// TIA Portal V19 export
FUNCTION "M_CmpGTE" : Bool   // FC43, LAD
TITLE = Module compare GREATHER THAN EQUAL / Module compare Greater than equal
// stored: Access Published, SetENOAutomatically false
   VAR_INPUT
      Xa : LReal;
      Xb : LReal;
      MODULE : LReal;
   END_VAR
BEGIN

REGION Network 1 (SCL): Xa >= Xb return TRUE / Main
   #M_CmpGTE := "M_PosAMinusPosB"(PosA := #Xa, PosB := #Xb, MODULE := #MODULE) >= 0.0;
END_REGION
END_FUNCTION
